// TIA Portal V20 export
TYPE "LKinCtrl_Utilities_typeFocusSelectionConfiguration"
// stored: Access Published
   STRUCT
      selectedField { ExternalAccessible := 'False'; ExternalVisible := 'False'; ExternalWritable := 'False'} : Int;   // Lower bound of the array to be displayed in the table window.
   END_STRUCT;
END_TYPE
